DATA_BLOCK "DB_SCALE_CS_2"
{ S7_Optimized_Access := 'FALSE' }
VERSION : 0.0
"UDT_SIWA_CS"

BEGIN
   i_DB_Lenght := 222;
   i_MaxLifeBitCyc := 500;
   i_SFC_ERR_C := 16#0000;
   i_CMD_INPUT := 230;
   bo_CMD_TRIGGER := TRUE;
   bo_CMD_IN_PROGRESS := TRUE;
   bo_CMD_FINISHED_OK := FALSE;
   bo_CMD_ERR := FALSE;
   b_CMD_ERR_CODE := 16#00;
   i_PRESET_TARE := 0;
   b_SELECT_PROC_VAL := 16#00;
   b_SELECTED_PROC_VAL := 16#00;
   i_PROCESS_VALUE := -25;
   b_INFO_REFRESH_COUNT := 16#07;
   w_SCALE_STATUS := 16#02C0;
   b_OPR_ERR_MSG := 16#00;
   bo_FB_ERR := FALSE;
   b_FB_ERR_CODE := 16#00;
   bo_START_UP_IN_PROGRESS := FALSE;
   w_DB_RES92 := 16#0000;
   w_DB_RES93 := 16#0000;
   w_DB_RES94 := 16#0000;
   w_DB_RES95 := 16#0000;
   w_DB_RES96 := 16#0000;
   w_DB_RES97 := 16#0000;
   w_INT_USE := 16#0000;
   s_JUST_DAT.w_CALIB_DIGITS0 := 16#0000;
   s_JUST_DAT.w_CALIB_DIGITS1 := 16#EA60;
   s_JUST_DAT.w_CALIB_DIGITS2 := 16#0000;
   s_JUST_DAT.i_CALIB_WEIGHT1 := 2000;
   s_JUST_DAT.i_CALIB_WEIGHT2 := 0;
   s_JUST_DAT.b_SIGNAL_RANGE := 16#02;
   s_JUST_DAT.b_FILT_TYPE := 16#00;
   s_JUST_DAT.b_FILT_FREQ := 16#04;
   s_JUST_DAT.b_FILT_DEPTH := 16#0F;
   s_JUST_DAT.s_SCALE_ID := 'SIWAREX XX';
   s_JUST_DAT.i_MIN_WR := 20;
   s_JUST_DAT.i_MAX_WR := 2000;
   s_JUST_DAT.i_INCREMENT_WR := 1;
   s_JUST_DAT.i_WEIGHT_ST_STILL := 10;
   s_JUST_DAT.t_TIME_ST_STILL1 := T#1S;
   s_JUST_DAT.b_DEC_POINT := 16#02;
   s_JUST_DAT.b_ZERO_NEG_VALUE := 16#01;
   s_JUST_DAT.b_ZERO_POS_VALUE := 16#03;
   s_JUST_DAT.b_TARA_MAX := 16#64;
   s_JUST_DAT.i_Reserve := 0;
   s_JUST_DAT.s_LEGAL_TRADE := '----';
   s_JUST_DAT.s_WEGHT_UNIT := 'kg  ';
   s_LIMIT_PARA.i_LIMIT1_ON := 400;
   s_LIMIT_PARA.i_LIMIT1_OFF := 220;
   s_LIMIT_PARA.i_LIMIT2_ON := 1000;
   s_LIMIT_PARA.i_LIMIT2_OFF := 980;
   s_LIMIT_PARA.bo_LIMIT1_PARA := FALSE;
   s_LIMIT_PARA.bo_LIMIT2_PARA := FALSE;
   s_LIMIT_PARA.b_Reserve := 16#00;
   s_MODUL_INFO_DATA.s_MODUL_NAME := 'SIWAREX CS';
   s_MODUL_INFO_DATA.s_ORDER_NUM := '7MH4910-0AA01$00$00$00$00   ';
   s_MODUL_INFO_DATA.w_VERSION_HW := 16#0005;
   s_MODUL_INFO_DATA.s_VERSION_FW := 'V1.5';
   s_MODUL_INFO_DATA.w_CRC_CHECK := 16#0897;
   s_TARE_CONTROL.i_TARE_VALUE := 0;
   s_INTERNAL_PROC_VAL.w_CRC_CHECK := 16#0000;
   s_INTERNAL_PROC_VAL.b_Reserve := 16#00;
   s_INTERNAL_PROC_VAL.bo_PRESET_TARA := FALSE;
   s_INTERNAL_PROC_VAL.d_TARA_X_100 := 0;
   s_INTERNAL_PROC_VAL.d_ZERO_X_100 := 0;
   s_PROCESS_VALUES.w_CRC_CHECK := 16#9561;
   s_PROCESS_VALUES.bo_STA_WRI_PROT := FALSE;
   s_PROCESS_VALUES.bo_STA_WR_MIN := TRUE;
   s_PROCESS_VALUES.bo_STA_Reserve1 := FALSE;
   s_PROCESS_VALUES.bo_STA_Reserve2 := FALSE;
   s_PROCESS_VALUES.bo_STA_Reserve3 := FALSE;
   s_PROCESS_VALUES.bo_STA_Reserve4 := FALSE;
   s_PROCESS_VALUES.bo_STA_Reserve5 := FALSE;
   s_PROCESS_VALUES.bo_STA_ERROR_ON := FALSE;
   s_PROCESS_VALUES.bo_STA_LIMIT1_ON := FALSE;
   s_PROCESS_VALUES.bo_STA_LIMIT2_ON := FALSE;
   s_PROCESS_VALUES.bo_STA_TARED := FALSE;
   s_PROCESS_VALUES.bo_STA_TARED_BY_MANUAL := FALSE;
   s_PROCESS_VALUES.bo_STA_MAX_9E := FALSE;
   s_PROCESS_VALUES.bo_STA_025_D_ZERO := FALSE;
   s_PROCESS_VALUES.bo_STA_ST_STAND_SCALE_ON := TRUE;
   s_PROCESS_VALUES.bo_STA_SCALE_CALIBRATED := TRUE;
   s_PROCESS_VALUES.b_OPR_ERR_MSG := 16#00;
   s_PROCESS_VALUES.b_Reserve := 16#00;
   s_PROCESS_VALUES.i_GROSS_WEIGHT_PROC := -27;
   s_PROCESS_VALUES.i_NET_WEIGHT_PROC := -27;
   s_PROCESS_VALUES.i_TARE_WEIGHT_PROC := 0;
   s_PROCESS_VALUES.i_GROSS_NET_VALUE := -25;
   s_PROCESS_VALUES.d_GROSS_NET_VALUE_10X := -270;
   s_PROCESS_VALUES.i_TARE_VALUE := 0;
   s_PROCESS_VALUES.i_ADC_DIGIT := 9164;
   s_PROCESS_VALUES.i_ADC_DIGIT_FILTER := 9164;
   s_PROCESS_VALUES.s_WEIGHT_ASCII := 'B -     25 kg ';
   s_PROCESS_VALUES.i_MILISEC := 520;
   s_PROCESS_VALUES.b_SECONDS := 16#33;
   s_PROCESS_VALUES.b_MINUTE := 16#39;
   s_PROCESS_VALUES.i_HOURS := 57;
   i_DB_Lenght1 := 222;

END_DATA_BLOCK

